// Mitsubishi GX Works2 project: timer+counter+sequence_1   PLC: Q03UDV

PROGRAM MAIN
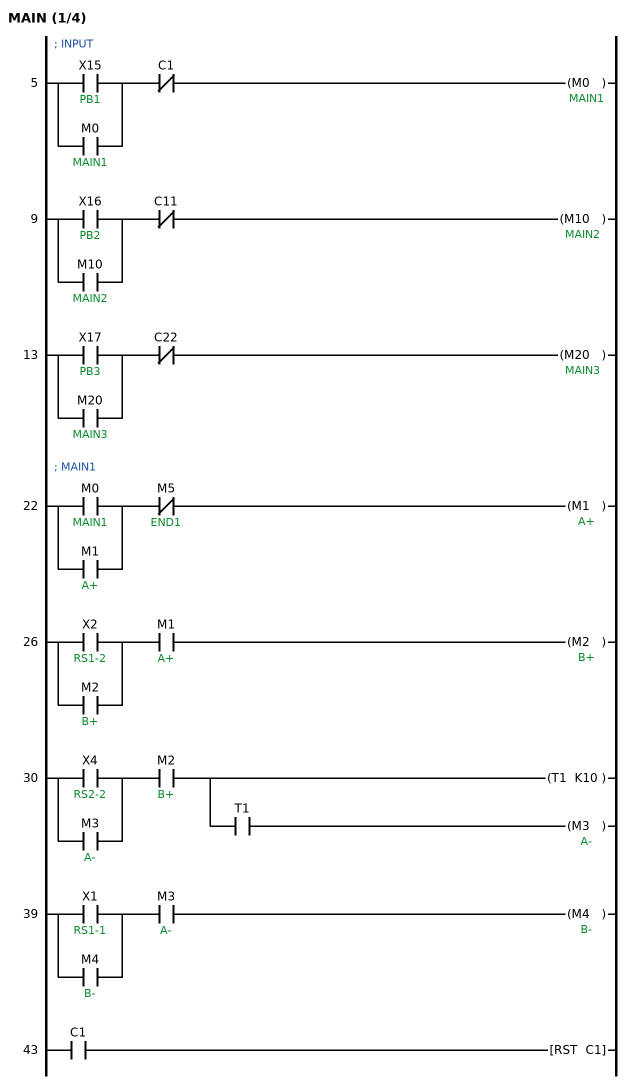
; INPUT
5     LD      X15  ; PB1
      OR      M0  ; MAIN1
      ANI     C1
      OUT     M0  ; MAIN1
9     LD      X16  ; PB2
      OR      M10  ; MAIN2
      ANI     C11
      OUT     M10  ; MAIN2
13    LD      X17  ; PB3
      OR      M20  ; MAIN3
      ANI     C22
      OUT     M20  ; MAIN3
; MAIN1
22    LD      M0  ; MAIN1
      OR      M1  ; A+
      ANI     M5  ; END1
      OUT     M1  ; A+
26    LD      X2  ; RS1-2
      OR      M2  ; B+
      AND     M1  ; A+
      OUT     M2  ; B+
30    LD      X4  ; RS2-2
      OR      M3  ; A-
      AND     M2  ; B+
      OUT     T1 K10
      AND     T1
      OUT     M3  ; A-
39    LD      X1  ; RS1-1
      OR      M4  ; B-
      AND     M3  ; A-
      OUT     M4  ; B-
43    LD      C1
      RST     C1
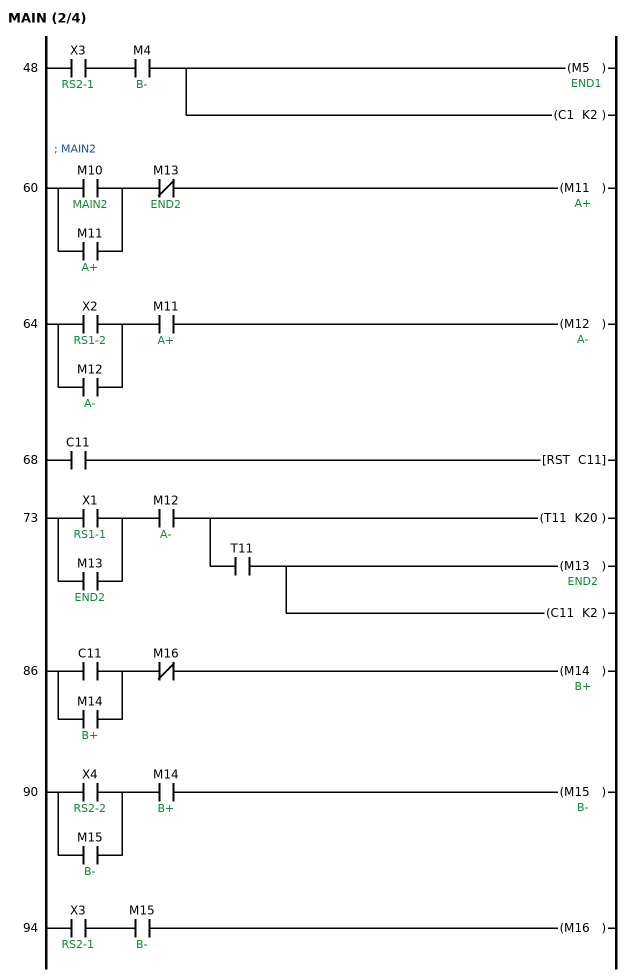
48    LD      X3  ; RS2-1
      AND     M4  ; B-
      OUT     M5  ; END1
      OUT     C1 K2
; MAIN2
60    LD      M10  ; MAIN2
      OR      M11  ; A+
      ANI     M13  ; END2
      OUT     M11  ; A+
64    LD      X2  ; RS1-2
      OR      M12  ; A-
      AND     M11  ; A+
      OUT     M12  ; A-
68    LD      C11
      RST     C11
73    LD      X1  ; RS1-1
      OR      M13  ; END2
      AND     M12  ; A-
      OUT     T11 K20
      AND     T11
      OUT     M13  ; END2
      OUT     C11 K2
86    LD      C11
      OR      M14  ; B+
      ANI     M16
      OUT     M14  ; B+
90    LD      X4  ; RS2-2
      OR      M15  ; B-
      AND     M14  ; B+
      OUT     M15  ; B-
94    LD      X3  ; RS2-1
      AND     M15  ; B-
      OUT     M16
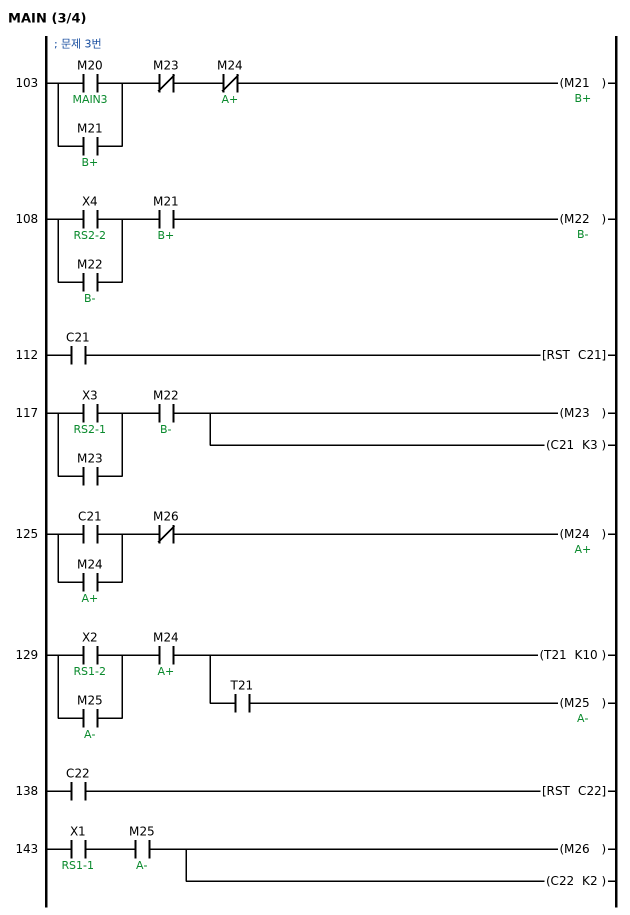
; 문제 3번
103   LD      M20  ; MAIN3
      OR      M21  ; B+
      ANI     M23
      ANI     M24  ; A+
      OUT     M21  ; B+
108   LD      X4  ; RS2-2
      OR      M22  ; B-
      AND     M21  ; B+
      OUT     M22  ; B-
112   LD      C21
      RST     C21
117   LD      X3  ; RS2-1
      OR      M23
      AND     M22  ; B-
      OUT     M23
      OUT     C21 K3
125   LD      C21
      OR      M24  ; A+
      ANI     M26
      OUT     M24  ; A+
129   LD      X2  ; RS1-2
      OR      M25  ; A-
      AND     M24  ; A+
      OUT     T21 K10
      AND     T21
      OUT     M25  ; A-
138   LD      C22
      RST     C22
143   LD      X1  ; RS1-1
      AND     M25  ; A-
      OUT     M26
      OUT     C22 K2
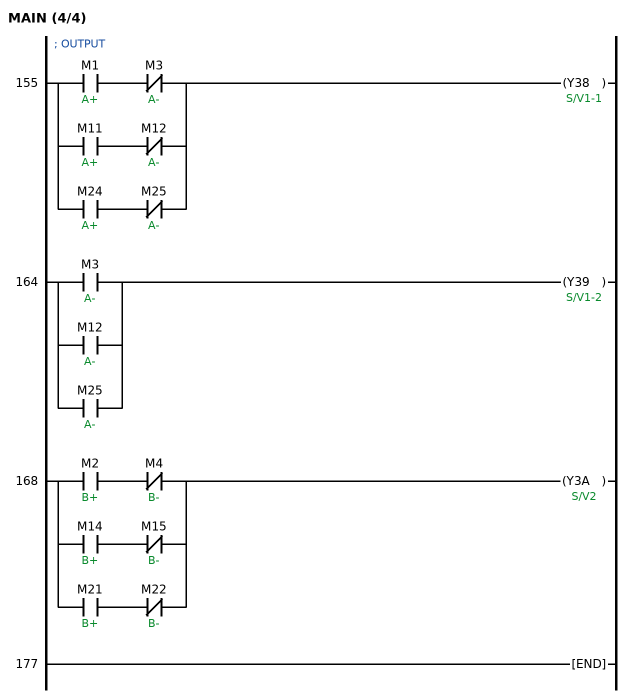
; OUTPUT
155   LD      M1  ; A+
      ANI     M3  ; A-
      LD      M11  ; A+
      ANI     M12  ; A-
      ORB
      LD      M24  ; A+
      ANI     M25  ; A-
      ORB
      OUT     Y38  ; S/V1-1
164   LD      M3  ; A-
      OR      M12  ; A-
      OR      M25  ; A-
      OUT     Y39  ; S/V1-2
168   LD      M2  ; B+
      ANI     M4  ; B-
      LD      M14  ; B+
      ANI     M15  ; B-
      ORB
      LD      M21  ; B+
      ANI     M22  ; B-
      ORB
      OUT     Y3A  ; S/V2
177   END
END_PROGRAM
